(* Logix 5000 project; controller cal1615 1756-L62 rev 20.19; software revision 20.05; part 16 of 81 *)
(* tags used below, declared in another part *)
   FAULT : BOOL;   // Fault AFI
   p01r09_pb_global_reset : BOOL;   // System Modes PB: Global Fault Reset
   p02r01 : routine;   // MOP HMI Iface Main
   p02r11 : routine;   // MOP HMI Iface
   p02r11_timer_fault : TIMER[4];   // MOP HMI Iface Fault Delay
   p02r11_timer_warning : TIMER[4];   // MOP HMI Iface Warning Delay
   p02r12 : routine;   // MOP HMI Iface
   p02r12_timer_fault : TIMER[4];   // MOP HMI Iface Fault Delay
   p02r12_timer_warning : TIMER[4];   // MOP HMI Iface Warning Delay
   p02r13 : routine;   // MOP HMI Iface
   p02r13_timer_fault : TIMER[4];   // MOP HMI Iface Fault Delay
   p02r13_timer_warning : TIMER[4];   // MOP HMI Iface Warning Delay
   p02r14 : routine;   // MOP HMI Iface
   p02r14_timer_fault : TIMER[4];   // MOP HMI Iface Fault Delay
   p02r14_timer_warning : TIMER[4];   // MOP HMI Iface Warning Delay
   p02r15 : routine;   // MOP HMI Iface
   p02r15_timer_fault : TIMER[4];   // MOP HMI Iface Fault Delay
   p02r15_timer_warning : TIMER[4];   // MOP HMI Iface Warning Delay
   p11r01 : routine;   // Zone 1 Main
(* P02_MOP_HMI_Iface, continued *)

ROUTINE R11   (* ladder *)
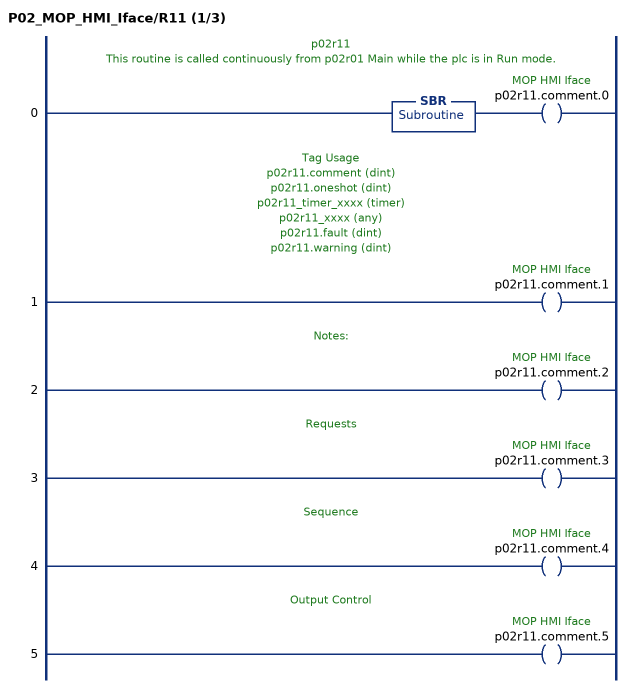
   // p02r11
   // This routine is called continuously from p02r01 Main while the plc is in Run mode.
   0: SBR()OTE(p02r11.comment.0);
   // Tag Usage
   // p02r11.comment (dint)
   // p02r11.oneshot (dint)
   // p02r11_timer_xxxx (timer)
   // p02r11_xxxx (any)
   // p02r11.fault (dint)
   // p02r11.warning (dint)
   1: OTE(p02r11.comment.1);
   // Notes:
   2: OTE(p02r11.comment.2);
   // Requests
   3: OTE(p02r11.comment.3);
   // Sequence
   4: OTE(p02r11.comment.4);
   // Output Control
   5: OTE(p02r11.comment.5);
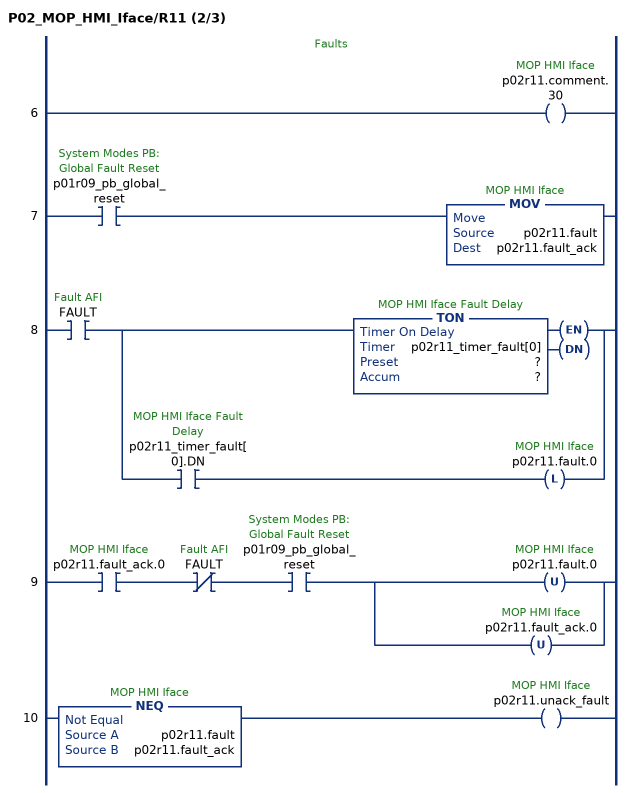
   // Faults
   6: OTE(p02r11.comment.30);
   7: XIC(p01r09_pb_global_reset)MOV(p02r11.fault,p02r11.fault_ack);
   8: XIC(FAULT)[TON(p02r11_timer_fault[0],?,?) ,XIC(p02r11_timer_fault[0].DN) OTL(p02r11.fault.0) ];
   9: XIC(p02r11.fault_ack.0)XIO(FAULT)XIC(p01r09_pb_global_reset)[OTU(p02r11.fault.0) ,OTU(p02r11.fault_ack.0) ];
   10: NEQ(p02r11.fault,p02r11.fault_ack)OTE(p02r11.unack_fault);
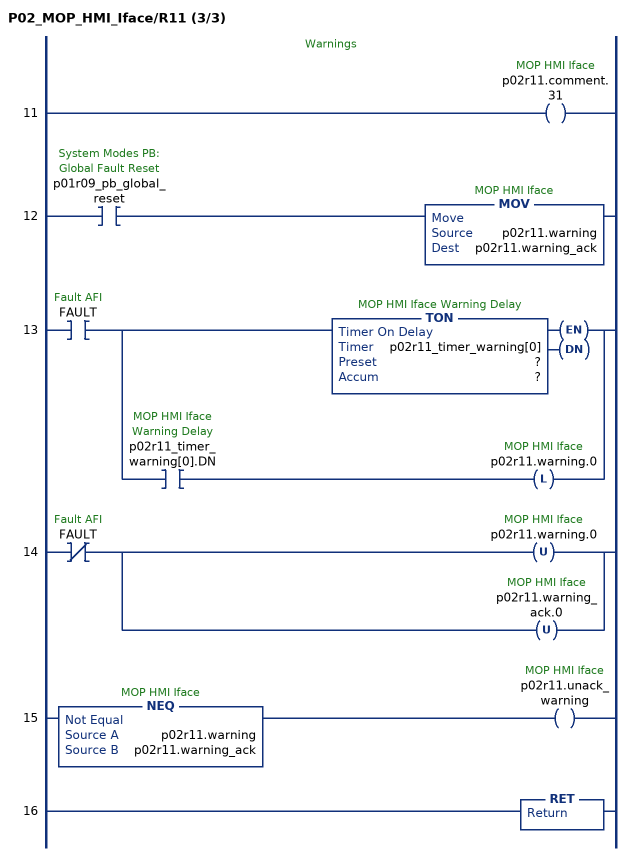
   // Warnings
   11: OTE(p02r11.comment.31);
   12: XIC(p01r09_pb_global_reset)MOV(p02r11.warning,p02r11.warning_ack);
   13: XIC(FAULT)[TON(p02r11_timer_warning[0],?,?) ,XIC(p02r11_timer_warning[0].DN) OTL(p02r11.warning.0) ];
   14: XIO(FAULT)[OTU(p02r11.warning.0) ,OTU(p02r11.warning_ack.0) ];
   15: NEQ(p02r11.warning,p02r11.warning_ack)OTE(p02r11.unack_warning);
   16: RET();
END_ROUTINE

ROUTINE R12   (* ladder *)
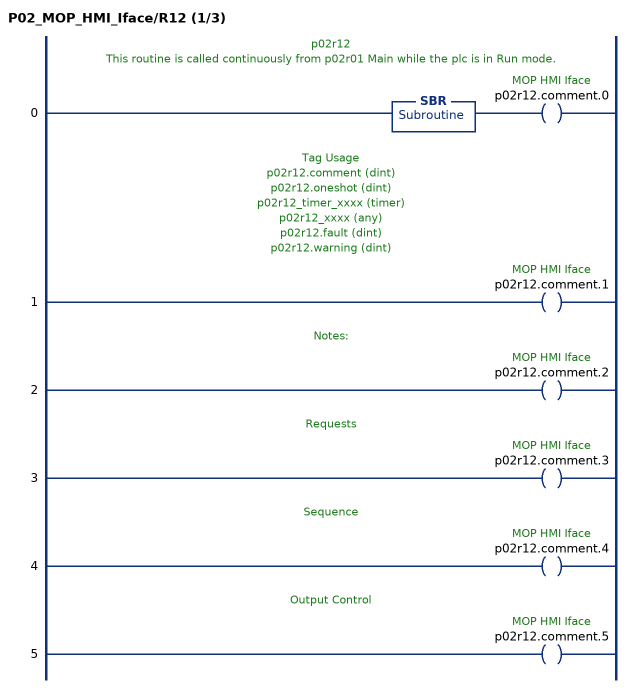
   // p02r12
   // This routine is called continuously from p02r01 Main while the plc is in Run mode.
   0: SBR()OTE(p02r12.comment.0);
   // Tag Usage
   // p02r12.comment (dint)
   // p02r12.oneshot (dint)
   // p02r12_timer_xxxx (timer)
   // p02r12_xxxx (any)
   // p02r12.fault (dint)
   // p02r12.warning (dint)
   1: OTE(p02r12.comment.1);
   // Notes:
   2: OTE(p02r12.comment.2);
   // Requests
   3: OTE(p02r12.comment.3);
   // Sequence
   4: OTE(p02r12.comment.4);
   // Output Control
   5: OTE(p02r12.comment.5);
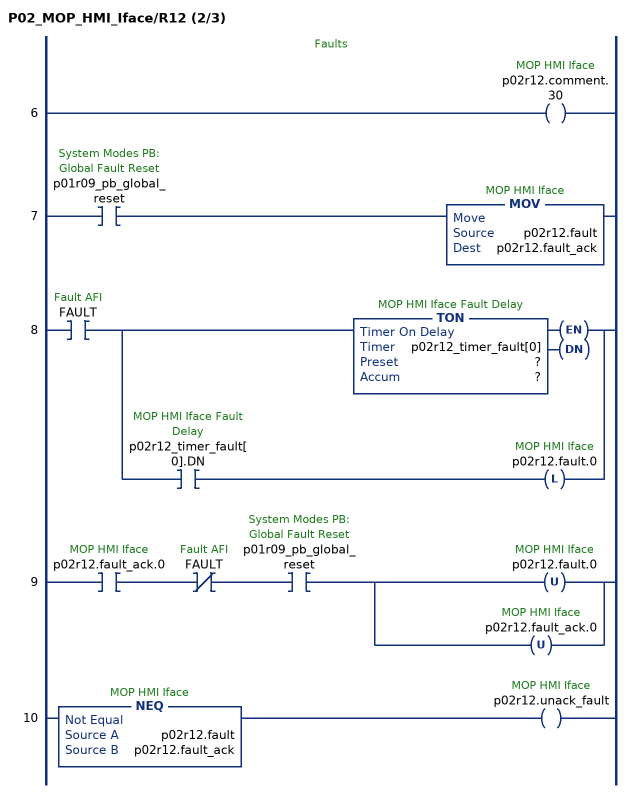
   // Faults
   6: OTE(p02r12.comment.30);
   7: XIC(p01r09_pb_global_reset)MOV(p02r12.fault,p02r12.fault_ack);
   8: XIC(FAULT)[TON(p02r12_timer_fault[0],?,?) ,XIC(p02r12_timer_fault[0].DN) OTL(p02r12.fault.0) ];
   9: XIC(p02r12.fault_ack.0)XIO(FAULT)XIC(p01r09_pb_global_reset)[OTU(p02r12.fault.0) ,OTU(p02r12.fault_ack.0) ];
   10: NEQ(p02r12.fault,p02r12.fault_ack)OTE(p02r12.unack_fault);
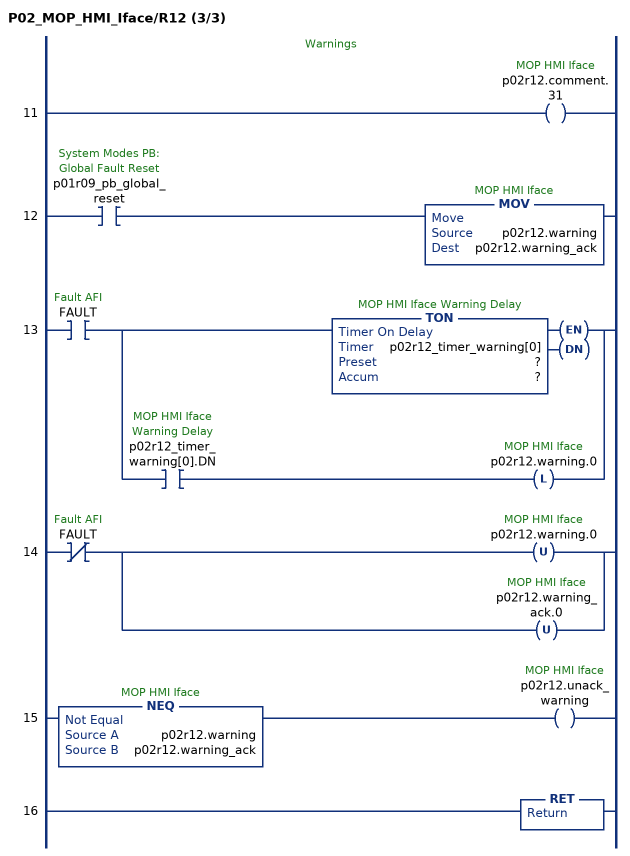
   // Warnings
   11: OTE(p02r12.comment.31);
   12: XIC(p01r09_pb_global_reset)MOV(p02r12.warning,p02r12.warning_ack);
   13: XIC(FAULT)[TON(p02r12_timer_warning[0],?,?) ,XIC(p02r12_timer_warning[0].DN) OTL(p02r12.warning.0) ];
   14: XIO(FAULT)[OTU(p02r12.warning.0) ,OTU(p02r12.warning_ack.0) ];
   15: NEQ(p02r12.warning,p02r12.warning_ack)OTE(p02r12.unack_warning);
   16: RET();
END_ROUTINE

ROUTINE R13   (* ladder *)
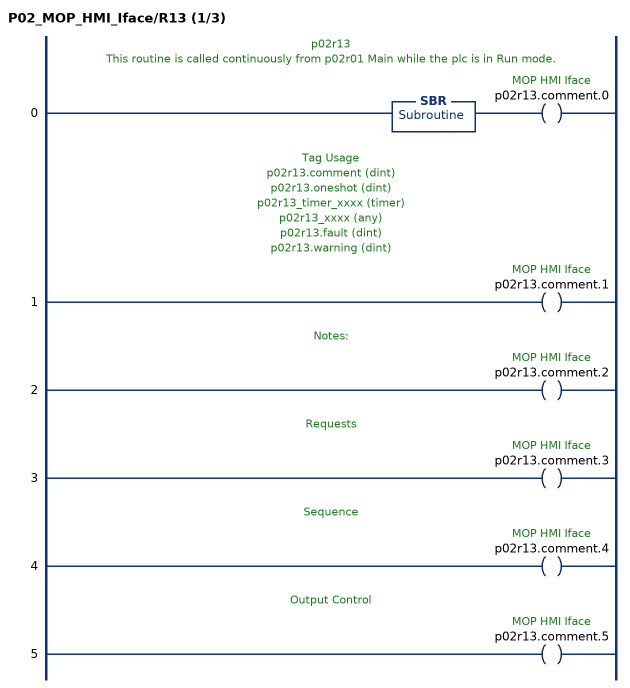
   // p02r13
   // This routine is called continuously from p02r01 Main while the plc is in Run mode.
   0: SBR()OTE(p02r13.comment.0);
   // Tag Usage
   // p02r13.comment (dint)
   // p02r13.oneshot (dint)
   // p02r13_timer_xxxx (timer)
   // p02r13_xxxx (any)
   // p02r13.fault (dint)
   // p02r13.warning (dint)
   1: OTE(p02r13.comment.1);
   // Notes:
   2: OTE(p02r13.comment.2);
   // Requests
   3: OTE(p02r13.comment.3);
   // Sequence
   4: OTE(p02r13.comment.4);
   // Output Control
   5: OTE(p02r13.comment.5);
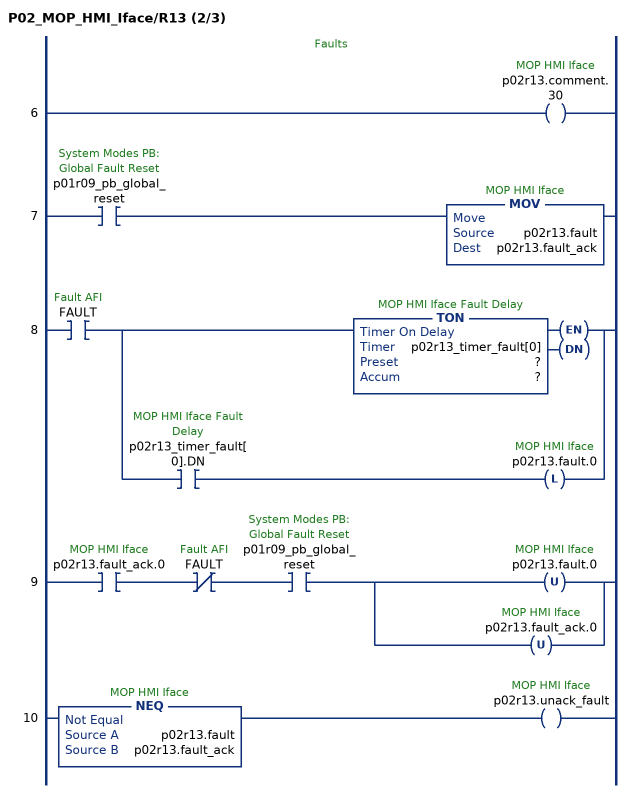
   // Faults
   6: OTE(p02r13.comment.30);
   7: XIC(p01r09_pb_global_reset)MOV(p02r13.fault,p02r13.fault_ack);
   8: XIC(FAULT)[TON(p02r13_timer_fault[0],?,?) ,XIC(p02r13_timer_fault[0].DN) OTL(p02r13.fault.0) ];
   9: XIC(p02r13.fault_ack.0)XIO(FAULT)XIC(p01r09_pb_global_reset)[OTU(p02r13.fault.0) ,OTU(p02r13.fault_ack.0) ];
   10: NEQ(p02r13.fault,p02r13.fault_ack)OTE(p02r13.unack_fault);
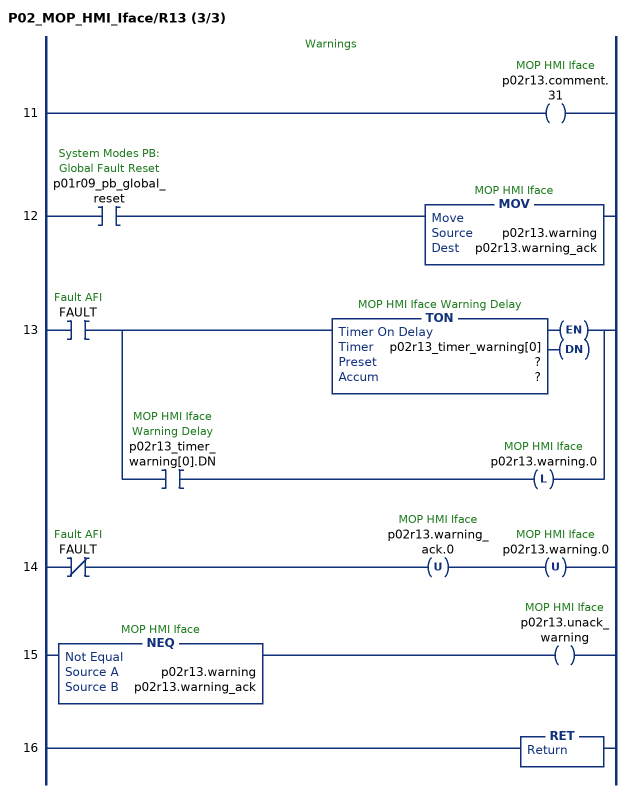
   // Warnings
   11: OTE(p02r13.comment.31);
   12: XIC(p01r09_pb_global_reset)MOV(p02r13.warning,p02r13.warning_ack);
   13: XIC(FAULT)[TON(p02r13_timer_warning[0],?,?) ,XIC(p02r13_timer_warning[0].DN) OTL(p02r13.warning.0) ];
   14: XIO(FAULT)OTU(p02r13.warning_ack.0)OTU(p02r13.warning.0);
   15: NEQ(p02r13.warning,p02r13.warning_ack)OTE(p02r13.unack_warning);
   16: RET();
END_ROUTINE

ROUTINE R14   (* ladder *)
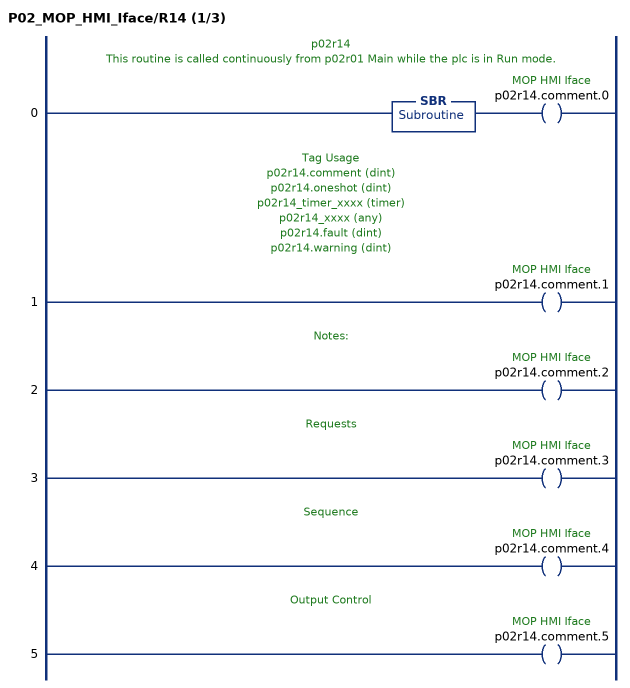
   // p02r14
   // This routine is called continuously from p02r01 Main while the plc is in Run mode.
   0: SBR()OTE(p02r14.comment.0);
   // Tag Usage
   // p02r14.comment (dint)
   // p02r14.oneshot (dint)
   // p02r14_timer_xxxx (timer)
   // p02r14_xxxx (any)
   // p02r14.fault (dint)
   // p02r14.warning (dint)
   1: OTE(p02r14.comment.1);
   // Notes:
   2: OTE(p02r14.comment.2);
   // Requests
   3: OTE(p02r14.comment.3);
   // Sequence
   4: OTE(p02r14.comment.4);
   // Output Control
   5: OTE(p02r14.comment.5);
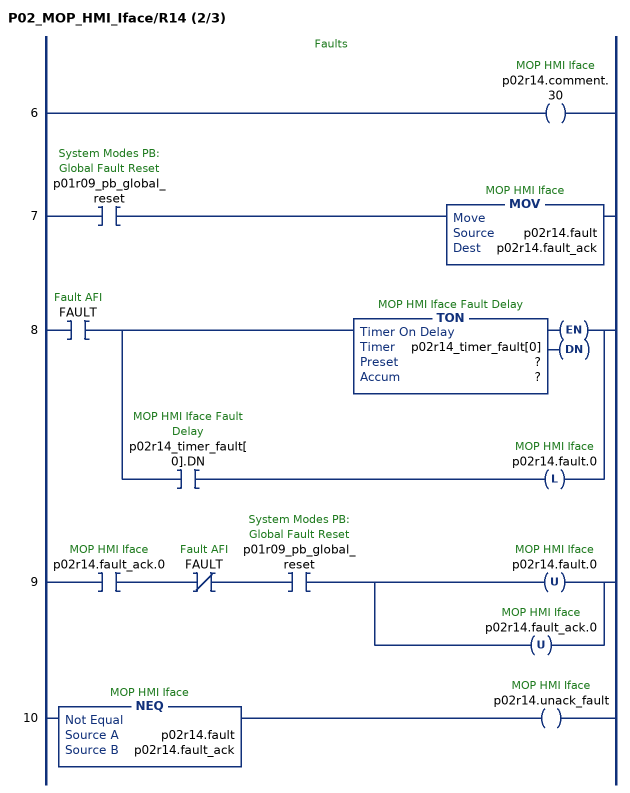
   // Faults
   6: OTE(p02r14.comment.30);
   7: XIC(p01r09_pb_global_reset)MOV(p02r14.fault,p02r14.fault_ack);
   8: XIC(FAULT)[TON(p02r14_timer_fault[0],?,?) ,XIC(p02r14_timer_fault[0].DN) OTL(p02r14.fault.0) ];
   9: XIC(p02r14.fault_ack.0)XIO(FAULT)XIC(p01r09_pb_global_reset)[OTU(p02r14.fault.0) ,OTU(p02r14.fault_ack.0) ];
   10: NEQ(p02r14.fault,p02r14.fault_ack)OTE(p02r14.unack_fault);
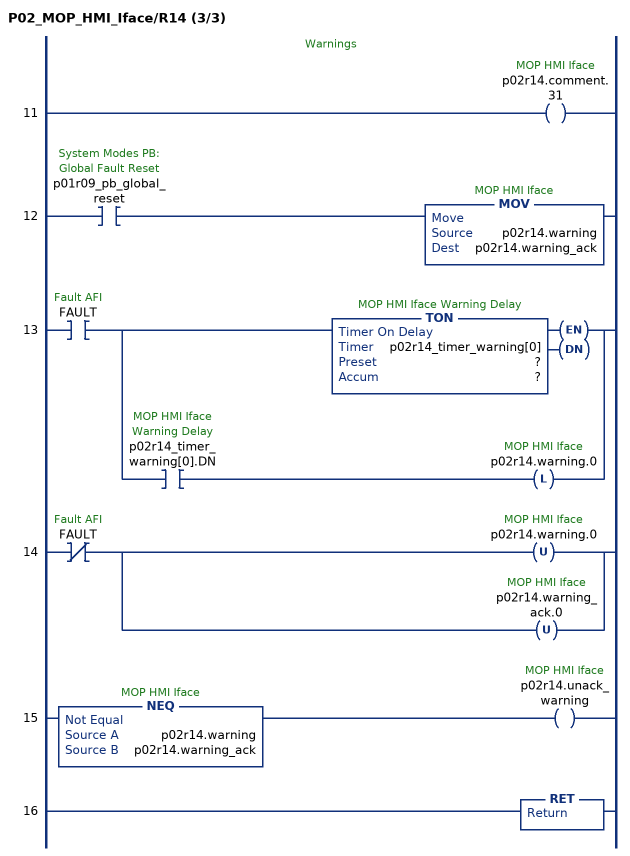
   // Warnings
   11: OTE(p02r14.comment.31);
   12: XIC(p01r09_pb_global_reset)MOV(p02r14.warning,p02r14.warning_ack);
   13: XIC(FAULT)[TON(p02r14_timer_warning[0],?,?) ,XIC(p02r14_timer_warning[0].DN) OTL(p02r14.warning.0) ];
   14: XIO(FAULT)[OTU(p02r14.warning.0) ,OTU(p02r14.warning_ack.0) ];
   15: NEQ(p02r14.warning,p02r14.warning_ack)OTE(p02r14.unack_warning);
   16: RET();
END_ROUTINE

ROUTINE R15   (* ladder *)
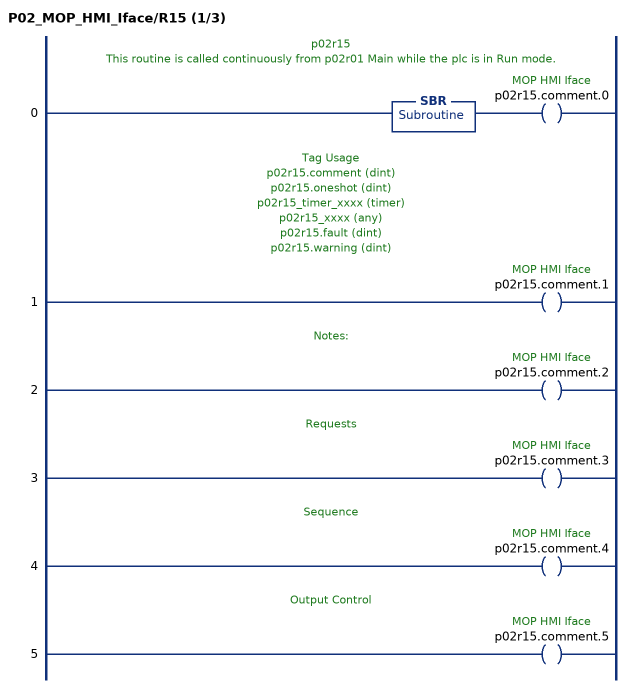
   // p02r15
   // This routine is called continuously from p02r01 Main while the plc is in Run mode.
   0: SBR()OTE(p02r15.comment.0);
   // Tag Usage
   // p02r15.comment (dint)
   // p02r15.oneshot (dint)
   // p02r15_timer_xxxx (timer)
   // p02r15_xxxx (any)
   // p02r15.fault (dint)
   // p02r15.warning (dint)
   1: OTE(p02r15.comment.1);
   // Notes:
   2: OTE(p02r15.comment.2);
   // Requests
   3: OTE(p02r15.comment.3);
   // Sequence
   4: OTE(p02r15.comment.4);
   // Output Control
   5: OTE(p02r15.comment.5);
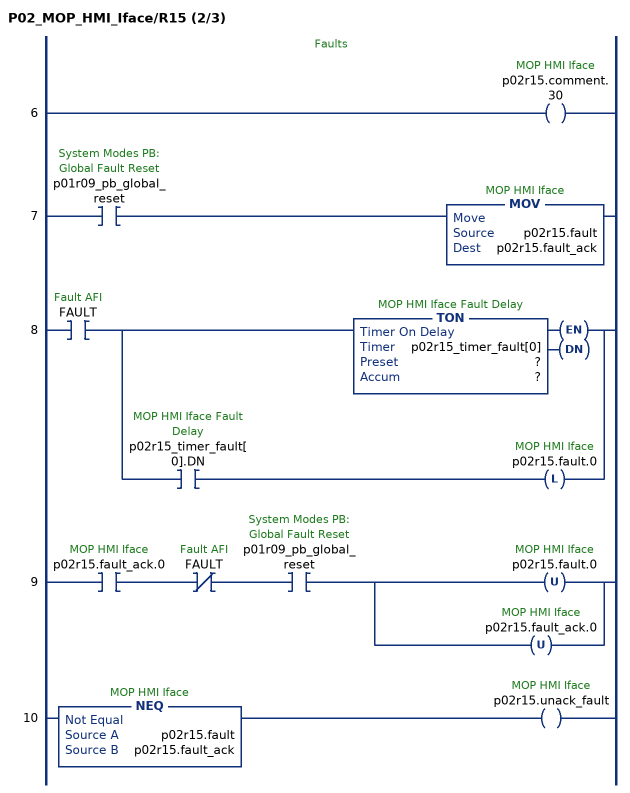
   // Faults
   6: OTE(p02r15.comment.30);
   7: XIC(p01r09_pb_global_reset)MOV(p02r15.fault,p02r15.fault_ack);
   8: XIC(FAULT)[TON(p02r15_timer_fault[0],?,?) ,XIC(p02r15_timer_fault[0].DN) OTL(p02r15.fault.0) ];
   9: XIC(p02r15.fault_ack.0)XIO(FAULT)XIC(p01r09_pb_global_reset)[OTU(p02r15.fault.0) ,OTU(p02r15.fault_ack.0) ];
   10: NEQ(p02r15.fault,p02r15.fault_ack)OTE(p02r15.unack_fault);
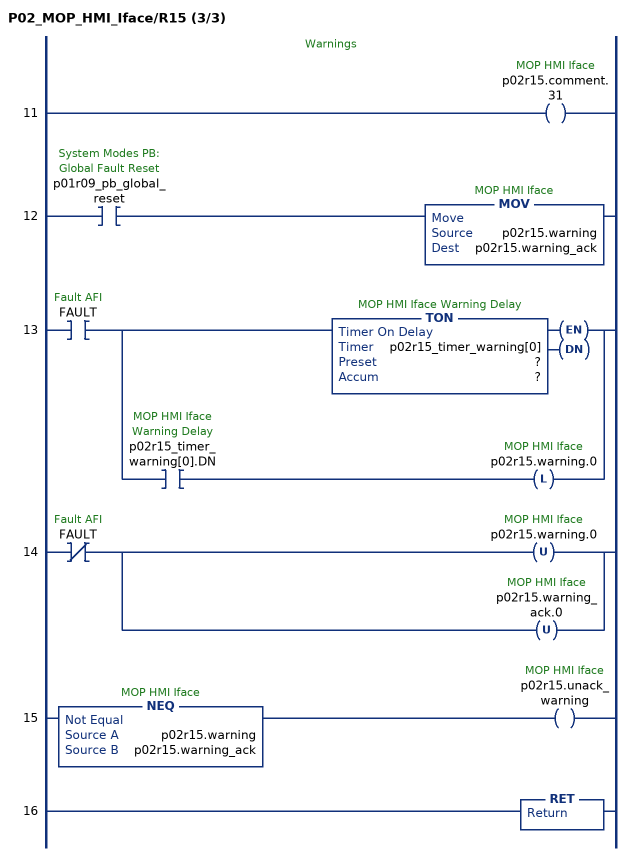
   // Warnings
   11: OTE(p02r15.comment.31);
   12: XIC(p01r09_pb_global_reset)MOV(p02r15.warning,p02r15.warning_ack);
   13: XIC(FAULT)[TON(p02r15_timer_warning[0],?,?) ,XIC(p02r15_timer_warning[0].DN) OTL(p02r15.warning.0) ];
   14: XIO(FAULT)[OTU(p02r15.warning.0) ,OTU(p02r15.warning_ack.0) ];
   15: NEQ(p02r15.warning,p02r15.warning_ack)OTE(p02r15.unack_warning);
   16: RET();
END_ROUTINE
END_PROGRAM

PROGRAM P11_Zone_1   (* main routine R01_Main *)

ROUTINE R01_Main   (* ladder *)
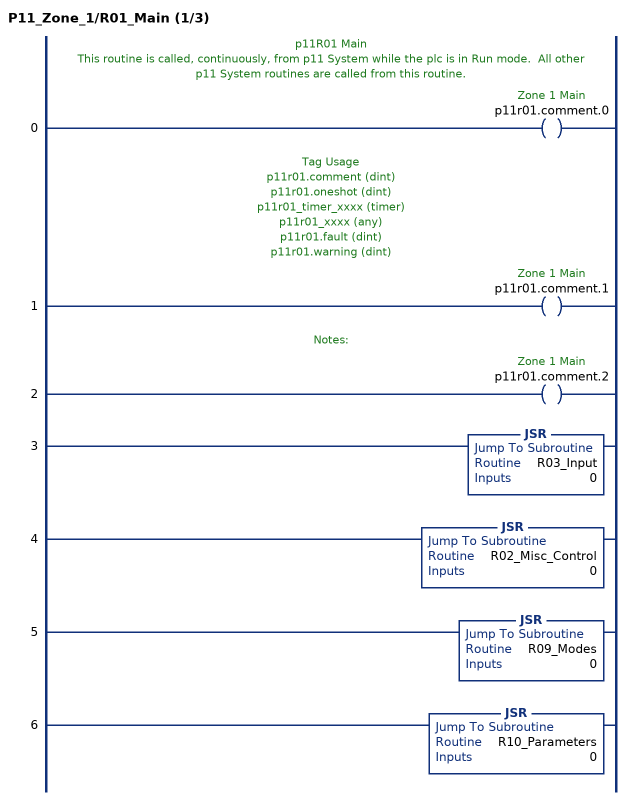
   // p11R01 Main
   // This routine is called, continuously, from p11 System while the plc is in Run mode.  All other p11 System routines are called from this routine.
   0: OTE(p11r01.comment.0);
   // Tag Usage
   // p11r01.comment (dint)
   // p11r01.oneshot (dint)
   // p11r01_timer_xxxx (timer)
   // p11r01_xxxx (any)
   // p11r01.fault (dint)
   // p11r01.warning (dint)
   1: OTE(p11r01.comment.1);
   // Notes:
   2: OTE(p11r01.comment.2);
   3: JSR(R03_Input,0);
   4: JSR(R02_Misc_Control,0);
   5: JSR(R09_Modes,0);
   6: JSR(R10_Parameters,0);
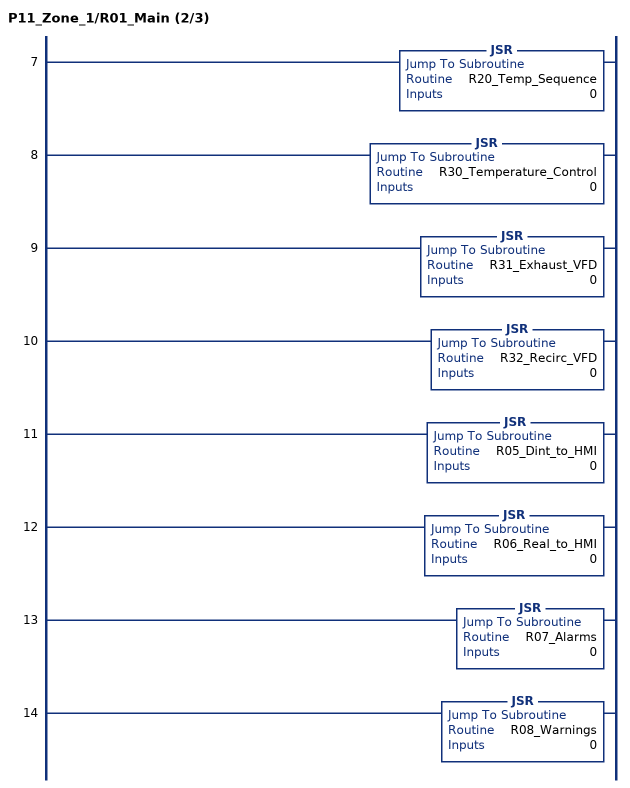
   7: JSR(R20_Temp_Sequence,0);
   8: JSR(R30_Temperature_Control,0);
   9: JSR(R31_Exhaust_VFD,0);
   10: JSR(R32_Recirc_VFD,0);
   11: JSR(R05_Dint_to_HMI,0);
   12: JSR(R06_Real_to_HMI,0);
   13: JSR(R07_Alarms,0);
   14: JSR(R08_Warnings,0);
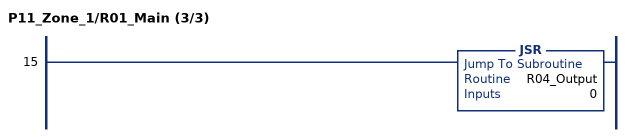
   15: JSR(R04_Output,0);
END_ROUTINE
